FUNCTION_BLOCK FB_CleaningProcessStateError EXTENDS FB_CleaningProcessStateBase
VAR_INPUT
END_VAR
VAR_OUTPUT
END_VAR
VAR
END_VAR

METHOD mAbort : BOOL
VAR_INPUT
END_VAR
IF NOT bL_DevOpActive THEN
  bL_DevOpActive := TRUE; //Set to relaunch process
  iL_CurrentStep := 0;
END_IF
I_ParentCallback.mSetMode(EN_Cleaning_OP.eOPEXITERROR);
I_ParentCallback.mDeviceAbort();
END_METHOD

METHOD mAckError : BOOL
VAR_INPUT
END_VAR

VAR
	sL_DeviceStatus: ST_CLEANING_DEV_STATUS;
END_VAR
sL_DeviceStatus := I_ParentCallback.pDeviceStatus;

IF NOT sL_DeviceStatus.bError THEN
  IF NOT SUPER^.pInitDone THEN
    I_ParentCallback.mChangeState(EN_Cleaning_State.Init);
  ELSE  
    I_ParentCallback.mChangeState(EN_Cleaning_State.Service);
  END_IF
END_IF
END_METHOD

METHOD mStateAction
VAR_INPUT
END_VAR

VAR
	sL_DeviceStatus: ST_CLEANING_DEV_STATUS;
END_VAR
sL_DeviceStatus := I_ParentCallback.pDeviceStatus;

SUPER^.pInitDone := sL_DeviceStatus.bRefKnown;

IF bL_DevOpActive THEN
	mDevOp();
END_IF
END_METHOD

END_FUNCTION_BLOCK

(* stored: Version 1.1.0.1, ProductVersion 3.1.4024.11
   POU FB_CleaningProcessStateError: Id {88ff0672-26ba-4329-bfb3-65ec1ae93a52}, SpecialFunc None
   Method mAbort: Id {6e20911d-6b5a-47ca-9e83-6d2d980dcf59}
   Method mAckError: Id {2be7c66b-44e5-4a17-8c7e-135a3c45d3f4}
   Method mStateAction: Id {a6f54142-1b86-4888-9377-9e0e666ff071} *)
